FUNCTION_BLOCK FB_UpdateStatus 
VAR_INPUT
	iLevel:UINT;
END_VAR
VAR
	EmptyEvents: ST_Event; // to Clear the event array[n]
	stManualBtnEvent:ST_Event;
	CmdEmpty: ST_Command;
	//i: UINT;            //temporary variable to loop all 6 parameters
	bErr: BOOL;         //temporary var for error flag
	sStatus:STRING;     //temporary var for error message

	sLogName: STRING(255);
	iEventName: E_EventName;
	sEventName: STRING(81);
	iSendEvent: UINT;
	eModuleID : E_ModuleID;
	
	//user pause button press event
	//RS_LanePause: RS;
	rtRiseBtn1Trig : R_Trig;
	ftFallBtn1Trig : F_Trig;	
	Btn1Tim: Ton;
	
	rtRiseBtn2Trig : R_Trig;
	ftFallBtn2Trig : F_Trig;	
	Btn2Tim: Ton;
	
	rtRiseBtn3Trig : R_Trig;
	ftFallBtn3Trig : F_Trig;	
	Btn3Tim: Ton;
	
	rtRiseBtn5Trig : R_Trig;
	ftFallBtn5Trig : F_Trig;	
	Btn5Tim: Ton;
	
	sentManualBtnEvent:bool;

	// DoorRecStarted
	//rtDoorRecStarted:R_Trig;
	
	
	//user load button press event	
	rtRiseTrig : R_Trig;
	ftFallTrig : F_Trig;
	LoadPbDly: Ton;
	tim:TON;
	
	sMessage : STRING;
	
	
//	[Step Mode]
	bPrevStepMode : ARRAY [1..NO_OF_LEVEL] OF BOOL;
	rtStep     : ARRAY[1..NO_OF_LEVEL] OF R_TRIG ;
	stPOCVIO   : ST_TCShuttlePOC_VIO;
	stMLVIO   : ST_TCMultiLevel_VIO;
	sStepMode : ARRAY[0..1] OF STRING := ['Off', 'On'];	
//	[Diagnostic Mode]
	bPrevDiagnosticMode:BOOL;
	
	stColVIO : ST_TCColumn_VIO;
	EmptyAlmStructure : ST_AlarmModules;
	
	i:INT;
	fbButtonBlinkTest:  FB_Blink;
	iButtonBlinkTest:INT;
	bButtonBlinkTest:BOOL;
	fbButtonBlinks:ARRAY [1..NO_OF_LEVEL,0..NO_OF_BTNLED-1] OF  FB_Blink;
	//fbButtonBlinks: ARRAY [1..NO_OF_LEVEL,0..NO_OF_BTNLED] OF FB_Blink;
	bTriggerBlinks: ARRAY [1..NO_OF_LEVEL,0..NO_OF_BTNLED-1] OF BOOL;
	bLastTriggerBlinks: ARRAY [1..NO_OF_LEVEL,0..NO_OF_BTNLED-1] OF BOOL;
	iBtnMode:ARRAY [1..NO_OF_LEVEL,0..NO_OF_BTNLED-1] OF INT;
	eLED:E_LED;
	iBtnLEDModes:ARRAY[1..NO_OF_LEVEL,0..NO_OF_BTNLED-1] OF INT;	// Created 2 dim array to check busy mode for indvidual mode
	iBtnLEDModeStatus:ARRAY[1..NO_OF_LEVEL,0..NO_OF_BTNLED-1] OF INT;
	tBlinkDuration:TIME:=T#1000MS;
	iFreq:DINT;
	bState:BOOL;
	
	
END_VAR

//[Set Pwr On Checkdelay from HMI]
	IF BtnSetTstPwrOnChkDelay AND iTstPwrOnChkDelay>=0 THEN 
		TstPwrOnChkDelay										:= INT_TO_TIME(iTstPwrOnChkDelay);
		BtnSetTstPwrOnChkDelay									:= FALSE;
	END_IF
	
	IF BtnSetAPPwrOnChkDelay AND iAPPwrOnChkDelay>=0 THEN 
		APPwrOnChkDelay											:= INT_TO_TIME(iAPPwrOnChkDelay);
		BtnSetAPPwrOnChkDelay									:= FALSE;
	END_IF	
	
	IF BtnSetTstReadyCheckDelay AND iTstReadyCheckDelay>=0 THEN 
		TstReadyCheckDelay										:= INT_TO_TIME(iTstReadyCheckDelay);
		BtnSetTstReadyCheckDelay								:= FALSE;
	END_IF
	
	IF BtnSetAPReadyCheckDelay AND iAPReadyCheckDelay>=0 THEN 
		APReadyCheckDelay										:= INT_TO_TIME(iAPReadyCheckDelay);
		BtnSetAPReadyCheckDelay									:= FALSE;
	END_IF
  
	bColIODiagnosticsMode										:= bDiagnosticMode;
	arrIODiagnosticsMode[iLevel]								:= bDiagnosticMode;

//	[ResetDuringSystemReset]
	IF FALSE THEN
		IF arrTCMultiLevel[iLevel].stGblParam.bInitialise THEN    // Need to use different variable 
			arrTCMultiLevel[iLevel].fbTCMultiLevelSeq.P_ErrClear	:= TRUE;
			ALMTC													:= EmptyAlmStructure;
		END_IF
		IF arrTCShuttlePOC[iLevel].stGblParam.bInitialise THEN
			arrTCShuttlePOC[iLevel].fbTCShuttlePOCSeq.P_ErrClear	:= TRUE;
			ALMTC													:= EmptyAlmStructure;
		END_IF	
	END_IF
//

//<ManualButtonPressedEvnt>    1=MaintenanceBtn,2=AbortFlowBtn,3=DoorUnlockBtn)
	stMLVIO 														:= arrTCMultiLevel[iLevel].fbTCMultiLevelSeq.P_stTCMultiLevelVIO;
	Btn1Tim(in:=stMLVIO.ipDrawerMaintenanceModeBtn, pt:=T#5MS);
	rtRiseBtn1Trig(Clk:=Btn1Tim.Q);
	ftFallBtn1Trig(Clk:=Btn1Tim.Q);
	
	Btn2Tim(in:=stMLVIO.ipTCCellAbortFlowBtn, pt:=T#5MS);
	rtRiseBtn2Trig(Clk:=Btn2Tim.Q);
	ftFallBtn2Trig(Clk:=Btn2Tim.Q);
	
	Btn3Tim(in:=stMLVIO.ipTCCellDoorOpenReqBtn, pt:=T#5MS);
	rtRiseBtn3Trig(Clk:=Btn3Tim.Q);
	ftFallBtn3Trig(Clk:=Btn3Tim.Q);
	
	sentManualBtnEvent												:= FALSE;
	
	IF rtRiseBtn1Trig.Q THEN
		stManualBtnEvent.eEventName									:= E_EventName.ManualButtonPressCompleted;
		stManualBtnEvent.sLogName									:= 'MaintenanceButtonPressed';
		stManualBtnEvent.eModuleID									:= LevelModuleID[iLevel]; //COLUMN_NAME;//E_ModuleID.COLUMN_LA;
		stManualBtnEvent.iParam[1]									:= 1;
		sentManualBtnEvent											:= TRUE;
		
	ELSIF rtRiseBtn2Trig.Q THEN
		stManualBtnEvent.eEventName									:= E_EventName.ManualButtonPressCompleted;
		stManualBtnEvent.sLogName									:= 'AbortFlowButtonPressed';
		stManualBtnEvent.eModuleID									:= LevelModuleID[iLevel];//COLUMN_NAME;//E_ModuleID.COLUMN_LA;
		stManualBtnEvent.iParam[1]									:= 2;
		sentManualBtnEvent											:= TRUE;
		
	ELSIF rtRiseBtn3Trig.Q THEN
		stManualBtnEvent.eEventName									:= E_EventName.ManualButtonPressCompleted;
		stManualBtnEvent.sLogName									:= 'DoorUnlockButtonPressed';
		stManualBtnEvent.eModuleID									:= LevelModuleID[iLevel];//COLUMN_NAME;//E_ModuleID.COLUMN_LA;
		stManualBtnEvent.iParam[1]									:= 3;
		sentManualBtnEvent											:= TRUE;
		
	END_IF
	
	IF sentManualBtnEvent THEN
		iBtnLEDModes[iLevel,stManualBtnEvent.iParam[1]]				:= 3;	//Blink (set Local Btn Mode flag to busy)
		CmdAndEventProcess.fbCmdAndEventUpdate.M_AddEvent(
			sLogName		:= stManualBtnEvent.sLogName, 
			eEventName		:= stManualBtnEvent.eEventName, 
			eModuleID		:= stManualBtnEvent.eModuleID, 
			iParam			:= stManualBtnEvent.iParam,
			sParam			:= EmptyEvents.sParam, 
			bParam			:= EmptyEvents.bParam, 
			dParam			:= EmptyEvents.dParam,
			sFailReason		:= EmptyEvents.sFailReason
		);
		
		sentManualBtnEvent											:= FALSE;
	END_IF
	
	
	IF ftFallBtn1Trig.Q THEN
		Btn1Tim(in:=FALSE);
	ELSIF ftFallBtn2Trig.Q THEN
		Btn2Tim(in:=FALSE);
	ELSIF ftFallBtn3Trig.Q THEN	
		Btn3Tim(in:=FALSE);
	END_IF

//<ButtonLEDBlink>
	(*===========================================
	SOLID OFF 	::State=0, 	Frequency = Don’tCare
	SOLID ON 	::State=1,	Frequency = 0
	BLINKING  	::State=1, 	Frequency = BlinkFreq
	===========================================*)

	//internal btn Status Adaptor between TA btn Blink Mode and FB_Blink Function Call
	FOR i:=0 TO NO_OF_BTNLED-1 DO   
		stMLVIO 									:= arrTCMultiLevel[iLevel].fbTCMultiLevelSeq.P_stTCMultiLevelVIO;
		
		CASE i OF     
			0 :	
				bState				:= stMLVIO.bMtnBtnLEDState;
				iFreq				:= stMLVIO.iMtnBtnLEDBlinkFreq;
			1 :	
				bState				:= stMLVIO.bAbtBtnLEDState;
				iFreq				:= stMLVIO.iAbtBtnLEDBlinkFreq;
			2 :	
				bState				:= stMLVIO.bDoorUnlockBtnLEDState;
				iFreq				:= stMLVIO.iDoorUnlockBtnLEDBlinkFreq;
		END_CASE
		
		IF (NOT bState) THEN
			iBtnLEDModes[iLevel,i]			:= 1;	//OFF,ON,BLINK
		ELSE
			IF iFreq <= 0 THEN
				//ONLED
				iBtnLEDModes[iLevel,i]		:= 2;
				
			ELSE
				//BLINK WITH BLINK RATE
				iBtnLEDModes[iLevel,i]		:= 3;
				tBlinkDuration				:= DINT_TO_TIME(iFreq);
			END_IF
		END_IF
	END_FOR

	FOR i:=0 TO NO_OF_BTNLED-1 DO
		//Converter for Button Blink Mode Status to TA 
		CASE iBtnLEDModes[iLevel,i] OF
			1 :	
				iBtnLEDModeStatus[iLevel,i]			:= 0 ;  //OFF
			2 :	
				iBtnLEDModeStatus[iLevel,i]			:= 2 ;  //ON
			3 :	
				iBtnLEDModeStatus[iLevel,i]			:= 1 ;  //BLINK
		END_CASE
		
		stMLVIO 									:= arrTCMultiLevel[iLevel].fbTCMultiLevelSeq.P_stTCMultiLevelVIO;
		fbButtonBlinks[iLevel,i](MODE:= iBtnLEDModes[iLevel,i], Duration:= tBlinkDuration, LED=> bTriggerBlinks[iLevel,i]);
		
		CASE i OF
			0 :	
				stMLVIO.opDrawerMaintenanceModeBtnLED		:= bTriggerBlinks[iLevel,i];
				stMLVIO.iMaintenanceButtonLEDStatusFlag 	:= iBtnLEDModeStatus[iLevel,i];
			1 :	
				stMLVIO.opTCCellAbortFlowBtnLED				:= bTriggerBlinks[iLevel,i];
				stMLVIO.iAbortButtonLEDStatusFlag			:= iBtnLEDModeStatus[iLevel,i];
			2 :	
				stMLVIO.opDoorOpenReqLED					:= bTriggerBlinks[iLevel,i];
				stMLVIO.iDoorLockButtonLEDStatusFlag		:= iBtnLEDModeStatus[iLevel,i];
		END_CASE
			
		IF bTriggerBlinks[iLevel,i] <> bLastTriggerBlinks[iLevel,i] THEN
			arrTCMultiLevel[iLevel].fbTCMultiLevelSeq.P_stTCMultiLevelVIO 		:= stMLVIO;
			bLastTriggerBlinks[iLevel,i] 										:= bTriggerBlinks[iLevel,i] ;
		END_IF
		
		IF stMLVIO.bOffBtnLeds[i] THEN
			iBtnLEDModes[iLevel,stManualBtnEvent.iParam[1]]						:= 1;
			arrTCMultiLevel[iLevel].fbTCMultiLevelSeq.P_stTCMultiLevelVIO 		:= stMLVIO;
			stMLVIO.bOffBtnLeds[i]												:= FALSE;
			arrTCMultiLevel[iLevel].fbTCMultiLevelSeq.P_stTCMultiLevelVIO 		:= stMLVIO;
		END_IF
	END_FOR
//</ButtonLEDBlink>

//	[DoorRecStartedEvnt]
	//rtDoorRecStarted(clk:=arrTCMultiLevel[iLevel].stGblParam.bDoorRecovery);
	IF arrTCMultiLevel[iLevel].stGblParam.bDoorRecoveryStarted OR arrTCShuttlePOC[iLevel].stGblParam.bDoorRecoveryStarted THEN
		tim(in:=TRUE,pt:=INT_TO_TIME(500));
		
		IF tim.Q THEN
			tim(in:=FALSE);
			CmdAndEventProcess.fbCmdAndEventUpdate.M_AddEvent( sLogName		:='DoorRecoveryStarted', 
															   eEventName	:= E_EventName.DoorRecoveryStarted, 
															   eModuleID	:= arrTCMultiLevel[iLevel].stGblParam.stDoorRecovEvnt.eModuleID, 
															   iParam		:= EmptyEvents.iParam, 
															   sParam		:= EmptyEvents.sParam, 
															   bParam		:= EmptyEvents.bParam, 
															   dParam		:= EmptyEvents.dParam, 
															   sFailReason	:= ''
			);
			
			arrTCMultiLevel[iLevel].stGblParam.bDoorRecoveryStarted				:= FALSE;
			arrTCMultiLevel[iLevel].stGblParam.bDoorRecovery					:= TRUE;
			arrTCShuttlePOC[iLevel].stGblParam.bDoorRecoveryStarted				:= FALSE;
			arrTCMultiLevel[iLevel].fbTCMultiLevelSeq.P_stParam 				:= arrTCMultiLevel[iLevel].stGblParam;
			arrTCShuttlePOC[iLevel].fbTCShuttlePOCSeq.P_stParam 				:= arrTCShuttlePOC[iLevel].stGblParam;
		END_IF
	END_IF
//--
//	[DoorRecoveryCompleted]
	IF arrTCMultiLevel[iLevel].stGblParam.bDoorRecoveryCompleted OR arrTCShuttlePOC[iLevel].stGblParam.bDoorRecoveryCompleted THEN 
		CmdAndEventProcess.fbCmdAndEventUpdate.M_AddEvent( sLogName		:= 'DoorRecoveryCompleted', 
														   eEventName	:= E_EventName.DoorRecoveryCompleted, 
														   eModuleID	:= arrTCMultiLevel[iLevel].stGblParam.stDoorRecovEvnt.eModuleID, 
														   iParam		:= EmptyEvents.iParam, 
														   sParam		:= EmptyEvents.sParam, 
														   bParam		:= EmptyEvents.bParam, 
														   dParam		:= EmptyEvents.dParam, 
														   sFailReason	:= ''
		);
		arrTCMultiLevel[iLevel].stGblParam.bDoorRecoveryCompleted:=FALSE;
		arrTCShuttlePOC[iLevel].stGblParam.bDoorRecoveryCompleted:=FALSE;
		arrTCMultiLevel[iLevel].fbTCMultiLevelSeq.P_stParam := arrTCMultiLevel[iLevel].stGblParam;
		arrTCShuttlePOC[iLevel].fbTCShuttlePOCSeq.P_stParam := arrTCShuttlePOC[iLevel].stGblParam;
	END_IF
//--
//	[DoorRecoveryFailed] //If DoorRecoveryFailed, Send Initialize Cmd.
	IF arrTCMultiLevel[iLevel].stGblParam.bDoorRecoveryFailed OR arrTCShuttlePOC[iLevel].stGblParam.bDoorRecoveryFailed THEN 
		CmdAndEventProcess.fbCmdAndEventUpdate.M_AddEvent( sLogName		:= 'DoorRecoveryFailed', 
														   eEventName	:= E_EventName.DoorRecoveryFailed, 
														   eModuleID	:= arrTCMultiLevel[iLevel].stGblParam.stDoorRecovEvnt.eModuleID, 
														   iParam		:= EmptyEvents.iParam, 
														   sParam		:= EmptyEvents.sParam, 
														   bParam		:= EmptyEvents.bParam, 
														   dParam		:= EmptyEvents.dParam, 
														   sFailReason	:= arrTCMultiLevel[iLevel].stGblParam.sFailReason
														   );
														   
		arrTCMultiLevel[iLevel].stGblParam.bDoorRecoveryFailed			:= FALSE;
		arrTCShuttlePOC[iLevel].stGblParam.bDoorRecoveryFailed			:= FALSE;
		arrTCMultiLevel[iLevel].stGblParam.bDoorRecovery				:= FALSE;
		arrTCShuttlePOC[iLevel].stGblParam.bDoorRecovery				:= FALSE;
		arrTCMultiLevel[iLevel].fbTCMultiLevelSeq.P_stParam 			:= arrTCMultiLevel[iLevel].stGblParam;
		arrTCShuttlePOC[iLevel].fbTCShuttlePOCSeq.P_stParam 			:= arrTCShuttlePOC[iLevel].stGblParam;
	END_IF
//--	
//<StepMode>
	IF arrStepMode[iLevel].bStepMode <> bPrevStepMode[iLevel] THEN //write when there is a chg for true or false
			stMLVIO 														:= arrTCMultiLevel[iLevel].fbTCMultiLevelSeq.P_stTCMultiLevelVIO;
			stMLVIO.bBypassSingleMove 										:= NOT arrStepMode[iLevel].bStepMode;
			arrTCMultiLevel[iLevel].fbTCMultiLevelSeq.P_stTCMultiLevelVIO	:= stMLVIO;
		
		fbFormat(sFormat:= 'bStepMode=%s, ModuleID=Level%d', arg1:= F_String(sStepMode[BOOL_TO_INT(arrStepMode[iLevel].bStepMode)]), arg2:= F_UInt(iLevel),sOut=> sMessage );
		Logging.fbDebugLog.M_nLogger(iLogLevel:= Logging.fbDebugLog.P_iLogVerbosity, sSource:= 'UserTrigger' , sMessage:= sMessage);
		bPrevStepMode[iLevel] 		:= arrStepMode[iLevel].bStepMode;
	END_IF
	
	rtStep[iLevel](CLK:=arrStepMode[iLevel].bStep);
	
	IF(rtStep[iLevel].Q) THEN //write only when true  
			stMLVIO 														:= arrTCMultiLevel[iLevel].fbTCMultiLevelSeq.P_stTCMultiLevelVIO;
			stMLVIO.bStep 													:= arrStepMode[iLevel].bStep;
			arrTCMultiLevel[iLevel].fbTCMultiLevelSeq.P_stTCMultiLevelVIO 	:= stMLVIO;
		
		fbFormat(sFormat:= 'bStep=%s, ModuleID=Level%d', arg1:= F_String(sStepMode[BOOL_TO_INT(arrStepMode[iLevel].bStep)]), arg2:= F_UInt(iLevel),sOut=> sMessage );
		Logging.fbDebugLog.M_nLogger(iLogLevel:= Logging.fbDebugLog.P_iLogVerbosity, sSource:= 'UserTrigger' , sMessage:= sMessage);
		
		arrStepMode[iLevel].bStep											:= FALSE; //reset gblbStep after receive from TA 
	END_IF
//</StepMode>

//<IODiagnostic>
	IF bPrevDiagnosticMode <> arrIODiagnosticsMode[iLevel] THEN
		stMLVIO 														:= arrTCMultiLevel[iLevel].fbTCMultiLevelSeq.P_stTCMultiLevelVIO ;
		stMLVIO.bDiagnosticMode 										:= arrIODiagnosticsMode[iLevel];
		arrTCMultiLevel[iLevel].fbTCMultiLevelSeq.P_stTCMultiLevelVIO  	:= stMLVIO;
		
		//POC
		stPOCVIO 														:= arrTCShuttlePOC[iLevel].fbTCShuttlePOCSeq.P_stTCPocVIO ;
		stPOCVIO.bDiagnosticMode 										:= arrIODiagnosticsMode[iLevel];
		arrTCShuttlePOC[iLevel].fbTCShuttlePOCSeq.P_stTCPocVIO  		:= stPOCVIO;

		bPrevDiagnosticMode 											:= arrIODiagnosticsMode[iLevel];
	END_IF

END_FUNCTION_BLOCK

(* stored: Version 1.1.0.1, ProductVersion 3.1.4022.18
   POU FB_UpdateStatus: Id {83131197-5d33-42fb-8f89-8ed06a50bc74}, SpecialFunc None *)
